PROGRAM EIP
VAR
	eip_input AT%I* 	: ARRAY[0..63] OF BYTE;
	eip_output AT%Q* 	: ARRAY[0..63] OF BYTE;
	
	i :UINT;
	counter : UINT;
	diff : BYTE;
END_VAR

IF counter > 255 THEN
	counter := 0;
ELSE
	counter := counter + 1;
END_IF

FOR i := 0 TO 63 DO
	eip_output[i] := UINT_TO_BYTE(counter);
END_FOR

diff := eip_output[1] - eip_input[1];

END_PROGRAM

(* stored: Version 1.1.0.1, ProductVersion 3.1.4024.12
   POU EIP: Id {c4a01dec-e004-4c77-adbe-3b40a0c27822}, SpecialFunc None *)
